ABB RobotStudio station: LAB1_29_08_20220831-101431.rsstn

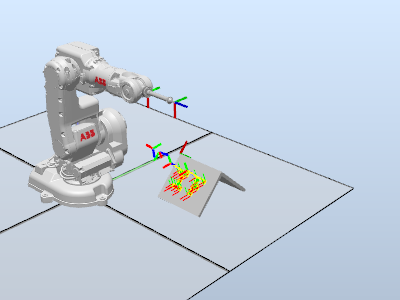
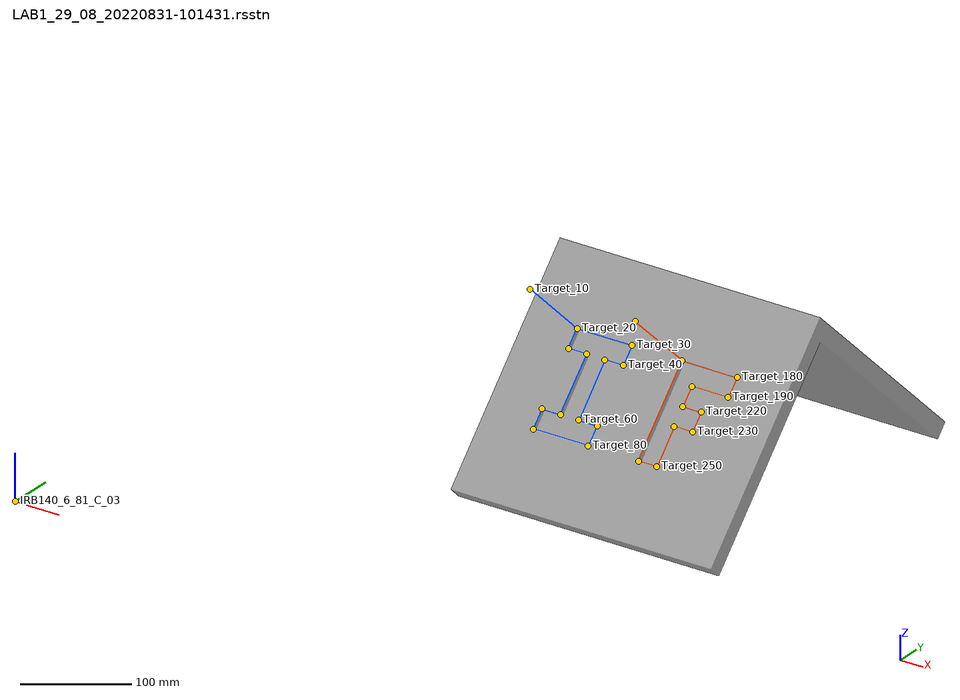
[picture v1: parts stored in the station drawn from their meshes, with robot base, taught points and paths (robot models come from the ABB library and are not in the file)]
Station LAB1_29_08 (saved by RobotStudio 22.2.9947.0)
Controller IRB140_6_81_1_LAB1_2908
  mechanical unit ROB_1: IRB140_6_81_C_03, 6 joints, base frame (0, 0, 0) mm
Layout (positions relative to the parent item):
  - IRB140_6_81_C_03 [mechanism, from Robots\IRB140_6_81_C_G_03.rslib] at (0, 0, 0) mm; joint values [0, 0, 0, 0, 0, 0] (rad or m)
  - workObjectIF [part] at (600, 400, 191.5) mm, rotated rx -137 ry 0 rz 180 deg, size 284.5 x 267 x 250 mm
  - marcadorIvandidas [mechanism] at (515, 0, 712) mm, rotated rx 0 ry 90 rz 0 deg
      TCP marcadorIvandidas at (-4.09, 34.34, 33.7) mm
      links: tool
Attachment: marcadorIvandidas is attached to IRB140_6_81_C_03 / Link6
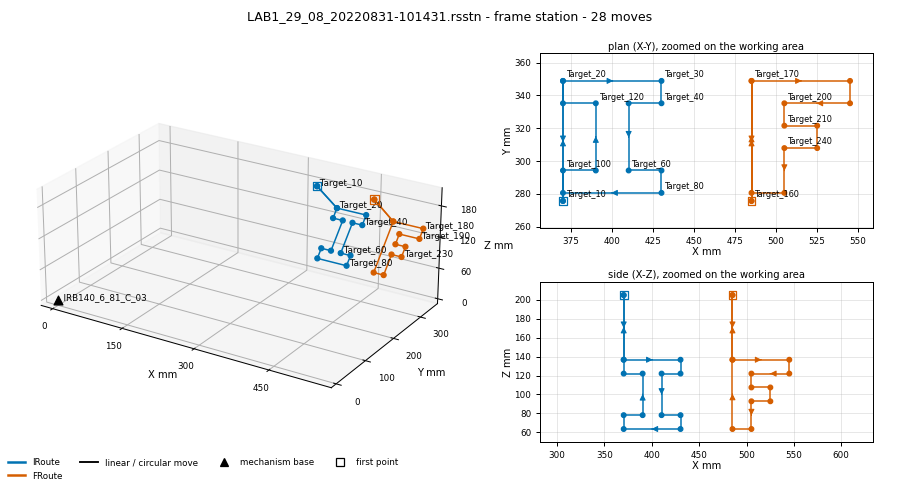
[picture p0: tool path of LAB1_29_08_20220831-101431.rsstn in frame station, 28 of 30 moves have a stored position in this frame; points joined in program order, loops and branches not executed]
Targets, tools, work objects and paths stored in the station, written as RAPID:
! task T_ROB1
MODULE CalibData
  PERS tooldata marcadorIvandidas:=[TRUE,[[0,0,164.8],[1,0,0,0]],[1,[0,0,1],[1,0,0,0],0,0,0]];
  TASK PERS wobjdata tableroIvandidas:=[FALSE,TRUE,"",[[0,0,0],[1,0,0,0]],[[315.5,400,191.5],[0.281957405,-0.64845973,-0.64845973,-0.281957405]]];
ENDMODULE

! task T_ROB1
MODULE Module1
  CONST robtarget Target_10:=[[-75.000236109,54.833333333,-99.999822919],[0.327947692,-0.000001116,0.000000387,-0.944695883],[0,0,-2,0],[9E+09,9E+09,9E+09,9E+09,9E+09,9E+09]];
  CONST robtarget Target_20:=[[-75,54.833333333,0.000177081],[0.327947692,-0.000001116,0.000000387,-0.944695883],[0,1,-2,0],[9E+09,9E+09,9E+09,9E+09,9E+09,9E+09]];
  CONST robtarget Target_30:=[[-75,114.833333333,0.000177081],[0.327947692,-0.000001116,0.000000387,-0.944695883],[0,0,-2,0],[9E+09,9E+09,9E+09,9E+09,9E+09,9E+09]];
  CONST robtarget Target_40:=[[-95,114.833333333,0.000224303],[0.327947692,-0.000001116,0.000000387,-0.944695883],[0,0,-2,0],[9E+09,9E+09,9E+09,9E+09,9E+09,9E+09]];
  CONST robtarget Target_50:=[[-95,94.833333333,0.000224303],[0.327947692,-0.000001116,0.000000387,-0.944695883],[0,0,-2,0],[9E+09,9E+09,9E+09,9E+09,9E+09,9E+09]];
  CONST robtarget Target_60:=[[-155,94.833333333,0.000365968],[0.327947692,-0.000001116,0.000000387,-0.944695883],[0,1,-2,0],[9E+09,9E+09,9E+09,9E+09,9E+09,9E+09]];
  CONST robtarget Target_70:=[[-155,114.833333333,0.000365968],[0.327947692,-0.000001116,0.000000387,-0.944695883],[0,0,-2,0],[9E+09,9E+09,9E+09,9E+09,9E+09,9E+09]];
  CONST robtarget Target_80:=[[-174.999999999,114.833333333,0.00041319],[0.327947692,-0.000001116,0.000000387,-0.944695883],[0,0,-2,0],[9E+09,9E+09,9E+09,9E+09,9E+09,9E+09]];
  CONST robtarget Target_90:=[[-174.999999999,54.833333333,0.00041319],[0.327947692,-0.000001116,0.000000387,-0.944695883],[0,1,-2,0],[9E+09,9E+09,9E+09,9E+09,9E+09,9E+09]];
  CONST robtarget Target_100:=[[-155,54.833333333,0.000365968],[0.327947692,-0.000001116,0.000000387,-0.944695883],[0,1,-2,0],[9E+09,9E+09,9E+09,9E+09,9E+09,9E+09]];
  CONST robtarget Target_110:=[[-155,74.833333333,0.000365968],[0.327947692,-0.000001116,0.000000387,-0.944695883],[0,1,-2,0],[9E+09,9E+09,9E+09,9E+09,9E+09,9E+09]];
  CONST robtarget Target_120:=[[-95,74.833333333,0.000224303],[0.327947692,-0.000001116,0.000000387,-0.944695883],[0,1,-2,0],[9E+09,9E+09,9E+09,9E+09,9E+09,9E+09]];
  CONST robtarget Target_130:=[[-95,54.833333333,0.000224303],[0.327947692,-0.000001116,0.000000387,-0.944695883],[0,1,-2,0],[9E+09,9E+09,9E+09,9E+09,9E+09,9E+09]];
  CONST robtarget Target_140:=[[-75,54.833333333,0.000177081],[0.327947692,-0.000001116,0.000000387,-0.944695883],[0,1,-2,0],[9E+09,9E+09,9E+09,9E+09,9E+09,9E+09]];
  CONST robtarget Target_150:=[[-75.000236109,54.833333333,-99.999822919],[0.327947692,-0.000001116,0.000000387,-0.944695883],[0,0,-2,0],[9E+09,9E+09,9E+09,9E+09,9E+09,9E+09]];
  CONST robtarget Target_160:=[[-75.000236109,169.666666667,-99.999822919],[0.327947692,-0.000001116,0.000000387,-0.944695883],[0,0,0,0],[9E+09,9E+09,9E+09,9E+09,9E+09,9E+09]];
  CONST robtarget Target_170:=[[-75,169.666666667,0.000177081],[0.327947692,-0.000001116,0.000000387,-0.944695883],[0,0,-2,0],[9E+09,9E+09,9E+09,9E+09,9E+09,9E+09]];
  CONST robtarget Target_180:=[[-75,229.666666667,0.000177081],[0.327947692,-0.000001116,0.000000387,-0.944695883],[0,0,-1,0],[9E+09,9E+09,9E+09,9E+09,9E+09,9E+09]];
  CONST robtarget Target_190:=[[-95,229.666666667,0.000224303],[0.327947692,-0.000001116,0.000000387,-0.944695883],[0,0,-2,0],[9E+09,9E+09,9E+09,9E+09,9E+09,9E+09]];
  CONST robtarget Target_200:=[[-95,189.666666667,0.000224303],[0.327947692,-0.000001116,0.000000387,-0.944695883],[0,0,-2,0],[9E+09,9E+09,9E+09,9E+09,9E+09,9E+09]];
  CONST robtarget Target_210:=[[-114.999999999,189.666666667,0.000271525],[0.327947692,-0.000001116,0.000000387,-0.944695883],[0,0,-2,0],[9E+09,9E+09,9E+09,9E+09,9E+09,9E+09]];
  CONST robtarget Target_220:=[[-114.999999999,209.666666667,0.000271525],[0.327947692,-0.000001116,0.000000387,-0.944695883],[0,0,-2,0],[9E+09,9E+09,9E+09,9E+09,9E+09,9E+09]];
  CONST robtarget Target_230:=[[-135,209.666666667,0.000318747],[0.327947692,-0.000001116,0.000000387,-0.944695883],[0,0,-2,0],[9E+09,9E+09,9E+09,9E+09,9E+09,9E+09]];
  CONST robtarget Target_240:=[[-135,189.666666667,0.000318747],[0.327947692,-0.000001116,0.000000387,-0.944695883],[0,0,-2,0],[9E+09,9E+09,9E+09,9E+09,9E+09,9E+09]];
  CONST robtarget Target_250:=[[-174.999999999,189.666666667,0.00041319],[0.327947692,-0.000001116,0.000000387,-0.944695883],[0,0,-2,0],[9E+09,9E+09,9E+09,9E+09,9E+09,9E+09]];
  CONST robtarget Target_260:=[[-174.999999999,169.666666667,0.00041319],[0.327947692,-0.000001116,0.000000387,-0.944695883],[0,0,-2,0],[9E+09,9E+09,9E+09,9E+09,9E+09,9E+09]];
  CONST robtarget Target_270:=[[-75,169.666666667,0.000177081],[0.327947692,-0.000001116,0.000000387,-0.944695883],[0,0,-2,0],[9E+09,9E+09,9E+09,9E+09,9E+09,9E+09]];
  CONST robtarget Target_280:=[[-75.000236109,169.666666667,-99.999822919],[0.327947692,-0.000001116,0.000000387,-0.944695883],[0,0,-1,0],[9E+09,9E+09,9E+09,9E+09,9E+09,9E+09]];
  CONST jointtarget Home:=[[0,0,0,0,0,0],[9E+09,9E+09,9E+09,9E+09,9E+09,9E+09]];
  CONST jointtarget MidPointViejo:=[[0,23.082008695,17.469851773,80.74339755,52.357742995,157.71972632],[9E+09,9E+09,9E+09,9E+09,9E+09,9E+09]];
  CONST jointtarget MidPoint:=[[0,20.632169141,9.010332751,11.163699287,62.137744693,0],[9E+09,9E+09,9E+09,9E+09,9E+09,9E+09]];
  PROC IRoute()
    MoveL Target_10,v200,fine,marcadorIvandidas\WObj:=tableroIvandidas;
    MoveL Target_20,v200,fine,marcadorIvandidas\WObj:=tableroIvandidas;
    MoveL Target_30,v200,fine,marcadorIvandidas\WObj:=tableroIvandidas;
    MoveL Target_40,v200,fine,marcadorIvandidas\WObj:=tableroIvandidas;
    MoveL Target_50,v200,fine,marcadorIvandidas\WObj:=tableroIvandidas;
    MoveL Target_60,v200,fine,marcadorIvandidas\WObj:=tableroIvandidas;
    MoveL Target_70,v200,fine,marcadorIvandidas\WObj:=tableroIvandidas;
    MoveL Target_80,v200,fine,marcadorIvandidas\WObj:=tableroIvandidas;
    MoveL Target_90,v200,fine,marcadorIvandidas\WObj:=tableroIvandidas;
    MoveL Target_100,v200,fine,marcadorIvandidas\WObj:=tableroIvandidas;
    MoveL Target_110,v200,fine,marcadorIvandidas\WObj:=tableroIvandidas;
    MoveL Target_120,v200,fine,marcadorIvandidas\WObj:=tableroIvandidas;
    MoveL Target_130,v200,fine,marcadorIvandidas\WObj:=tableroIvandidas;
    MoveL Target_140,v200,fine,marcadorIvandidas\WObj:=tableroIvandidas;
    MoveL Target_150,v200,fine,marcadorIvandidas\WObj:=tableroIvandidas;
  ENDPROC
  PROC FRoute()
    MoveL Target_160,v200,fine,marcadorIvandidas\WObj:=tableroIvandidas;
    MoveL Target_170,v200,fine,marcadorIvandidas\WObj:=tableroIvandidas;
    MoveL Target_180,v200,fine,marcadorIvandidas\WObj:=tableroIvandidas;
    MoveL Target_190,v200,fine,marcadorIvandidas\WObj:=tableroIvandidas;
    MoveL Target_200,v200,fine,marcadorIvandidas\WObj:=tableroIvandidas;
    MoveL Target_210,v200,fine,marcadorIvandidas\WObj:=tableroIvandidas;
    MoveL Target_220,v200,fine,marcadorIvandidas\WObj:=tableroIvandidas;
    MoveL Target_230,v200,fine,marcadorIvandidas\WObj:=tableroIvandidas;
    MoveL Target_240,v200,fine,marcadorIvandidas\WObj:=tableroIvandidas;
    MoveL Target_250,v200,fine,marcadorIvandidas\WObj:=tableroIvandidas;
    MoveL Target_260,v200,fine,marcadorIvandidas\WObj:=tableroIvandidas;
    MoveL Target_270,v200,fine,marcadorIvandidas\WObj:=tableroIvandidas;
    MoveL Target_280,v200,fine,marcadorIvandidas\WObj:=tableroIvandidas;
  ENDPROC
  PROC Homing()
    MoveAbsJ Home,v1000,z100,marcadorIvandidas\WObj:=tableroIvandidas;
  ENDPROC
  PROC MidPointGoing()
    MoveAbsJ MidPoint,v1000,z100,marcadorIvandidas\WObj:=tableroIvandidas;
  ENDPROC
ENDMODULE

